(* CoDeSys 2.3.5.6 project: lyjak_01_cfc.pro *)
(* Libraries: Standard.lib*4.1.15 17:23:13, SYSLIBCALLBACK.LIB*4.1.15 17:23:13 *)

(* PLC configuration (modules and I/O channels)
Configuration EC4P-200 [Root] node -1, in %IB0 out %QB0 {EC4P_RestartPwrOn = WARMSTART; EC4P_MaxCycleTime = 20; EC4P_Com1BaudRate = 38400; EC4P_CAN1BaudRate = 125KBaud; EC4P_RoutingId = 127; EC4P_EasyNetId = 1; EC4P_EasyNetCfg = 0; EC4P_EasyNetCycleTime = 50; EC4P_RoutingChannel = CAN1; EC4P_IPFlags = 0; EC4P_IPAddress = 0; EC4P_SubNetMask = 0; EC4P_DefaultGateway = 0; EC4P_SummerWinterFlags = 0; EC4P_SummerWinterRule1 = 0; EC4P_SummerWinterRule2 = 0}
  Local I/O [EC4P_LocalIO] node 0, in %IB0 out %QB0 {EC4P_LocalInt = 0}
    I1 AT %IX0.0 [LocalBitInput] Input I1
    I2 AT %IX0.1 [LocalBitInput] Input I2
    I3 AT %IX0.2 [LocalBitInput] Input I3
    I4 AT %IX0.3 [LocalBitInput] Input I4
    I5 AT %IX0.4 [LocalBitInput] Input I5
    I6 AT %IX0.5 [LocalBitInput] Input I6
    I7 AT %IX0.6 [LocalBitInput] Input I7
    I8 AT %IX0.7 [LocalBitInput] Input I8
    I9 AT %IX1.0 [LocalBitInput] Input I9
    I10 AT %IX1.1 [LocalBitInput] Input I10
    I11 AT %IX1.2 [LocalBitInput] Input I11
    I12 AT %IX1.3 [LocalBitInput] Input I12
    I13 AT %IX1.4 [LocalDiagInput] Diagnostic Input I13
    I14 AT %IX1.5 [LocalDiagInput] Diagnostic Input I14
    I15 AT %IX1.6 [LocalDiagInput] Diagnostic Input I15
    I16 AT %IX1.7 [LocalDiagInput] Diagnostic Input I16
    I7_Analog AT %IW2 [LocalAnalogIn] Input I7, 10Bit, 0-10VDC
    I8_Analog AT %IW4 [LocalAnalogIn] Input I8, 10Bit, 0-10VDC
    I11_Analog AT %IW6 [LocalAnalogIn] Input I11, 10Bit, 0-10VDC
    I12_Analog AT %IW8 [LocalAnalogIn] Input I12, 10Bit, 0-10VDC
    Transistor Outputs [EC4P_TOutputs] node 0, in %IB10 out %QB0
      Q1 AT %QX0.0 [LocalBitOutput] Transistor-Output Q1
      Q2 AT %QX0.1 [LocalBitOutput] Transistor-Output Q2
      Q3 AT %QX0.2 [LocalBitOutput] Transistor-Output Q3
      Q4 AT %QX0.3 [LocalBitOutput] Transistor-Output Q4
      Q5 AT %QX0.4 [LocalBitOutput] Transistor-Output Q5
      Q6 AT %QX0.5 [LocalBitOutput] Transistor-Output Q6
      Q7 AT %QX0.6 [LocalBitOutput] Transistor-Output Q7
      Q8 AT %QX0.7 [LocalBitOutput] Transistor-Output Q8
    No Analog Output [EC4P_NoAnalogOutput] node 1, in %IB10 out %QB1
    No Keys [EC4P_NoKeys] node 2, in %IB10 out %QB1
    No Counter [EC4P_NoCounter] node 3, in %IB10 out %QB1
  Extension [EC4P_Extension] node 1, in %IB10 out %QB1
    No Extension [EC4P_NoExtension] node 0, in %IB10 out %QB1
*)

(* POU PLC_PRG, CFC *)
PROGRAM PLC_PRG
VAR
END_VAR
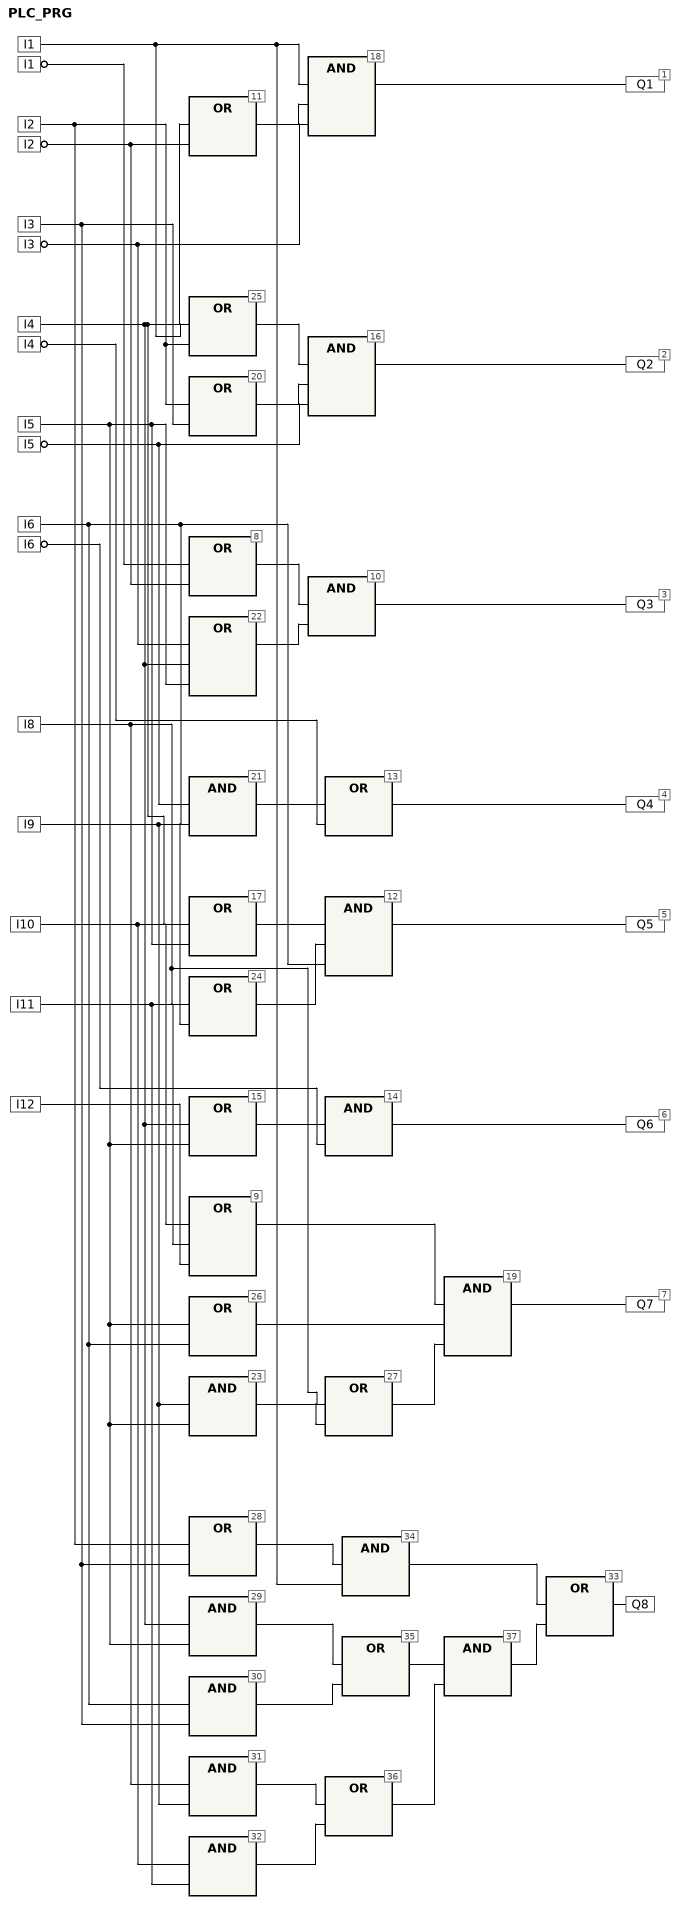
_CFC_ (* Continuous Function Chart, elements in execution order *)
#0 Q8 <= #33
#1 Q1 <= #18
#2 Q2 <= #16
#3 Q3 <= #10
#4 Q4 <= #13
#5 Q5 <= #12
#6 Q6 <= #14
#7 Q7 <= #19
#8 OR(NOT I1, NOT I2)
#9 OR(I10, I11, I12)
#10 AND(#8, #22)
#11 OR(I4, NOT I2)
#12 AND(#17, #24, I6)
#13 OR(#21, NOT I4)
#14 AND(#15, NOT I6)
#15 OR(I4, I5)
#16 AND(#25, #20, NOT I5)
#17 OR(I4, I5)
#18 AND(I1, #11, NOT I3)
#19 AND(#9, #26, #27)
#20 OR(I2, I3)
#21 AND(NOT I5, I6)
#22 OR(NOT I3, I4, I5)
#23 AND(I9, I5)
#24 OR(I8, I9)
#25 OR(I1, I2)
#26 OR(I5, I6)
#27 OR(I8, #23)
#28 OR(I2, I3)
#29 AND(I4, I5)
#30 AND(I6, I3)
#31 AND(I8, I9)
#32 AND(I10, I11)
#33 OR(#34, #37)
#34 AND(#28, I1)
#35 OR(#29, #30)
#36 OR(#31, #32)
#37 AND(#35, #36)
_END_CFC_
END_PROGRAM
